{attribute 'qualified_only'}
VAR_GLOBAL
	gCfg  : ST_DfiConfig;
	gDiag : ST_DfiDiag;
	// pipeline
	fbLoader  : FB_DfiConfigLoader;
	fbSub     : FB_DfiMqttSubscriber;
	fbParser  : FB_DfiPayloadParser;
	fbBuffer  : FB_DfiRowBuffer;
	fbSampler : FB_DfiSampler;
	fbWriter  : FB_DfiDbWriter;
END_VAR

(* stored: Version 1.1.0.1
   GVL GVL_Dfi: Id {dcd93ea1-13ee-404c-8c64-f1267f889f40} *)
